FUNCTION IsEmptyPort : BOOL
VAR_INPUT
	Port : I_Port;
END_VAR

IsEmptyPort := Port = 0;

END_FUNCTION

(* stored: Version 1.1.0.1, ProductVersion 3.1.4024.12
   POU IsEmptyPort: Id {ed526687-3cbe-0bbf-011b-976186cb0e13}, SpecialFunc None *)
